PROGRAM TestsBase
VAR
	CyclicRunner_TEST			   : CyclicRunner_TEST;
	ComponentCollection_TEST	   : ComponentCollection_TEST;
	Module_TEST					   : Module_TEST;
	CyclicComponent_TEST		   : CyclicComponent_TEST;
	Component_TEST				   : Component_TEST;
	ModuleCollection_TEST		   : ModuleCollection_TEST;
	Tracing_TEST				   : Tracing_TEST;
	Initializer_TEST			   : Initializer_TEST;
	Events_TEST					   : Events_TEST;
	Statemachine_TEST			   : Statemachine_TEST;
	Collection_Test				   : Collection_TEST();
	List_TEST					   : List_TEST;
	ModeControl_TEST			   : ModeControl_TEST;
	CollectionPeeker_Test		   : CollectionPeeker_Test;
	ForcibleBool_TEST			   : ForcibleBool_TEST;
	ForcibleInt_Test			   : ForcibleInt_Test;
	Utilities_TEST				   : Utilities_TEST;
	DigitalInput_NC_TEST		   : DigitalInput_NC_TEST;
	DigitalInput_NO_TEST		   : DigitalInput_NO_TEST;
	DigitalOutput_TEST			   : DigitalOutput_TEST;
	DigitalInput_Combiner_TEST	   : DigitalInput_Combiner_TEST;
	DigitalInput_Debounce_TEST	   : DigitalInput_Debounce_TEST;
	Cylinder_TEST				   : Cylinder_TEST;
	SafetyBase_TEST				   : SafetyBase_TEST;
	ADS_TEST					   : ADS_TEST;
	DigitalInput_ForceVisitor_TEST : DigitalInput_ForceVisitor_TEST;
	Recipe_TEST					   : Recipe_TEST;
	Analog_TEST					   : Analog_TEST;
	Serial_TEST					   : SerialConnection_Tests;
	Axis_Test					   : Axis_Test;
	EtherCatMaster_TEST		   : EtherCatMaster_TEST;

	//
	Component1				  : CyclicComponent_Mockup('Component 1');
	Component2				  : CyclicComponent_Mockup('Component 2');
	Component3				  : CyclicComponent_Mockup('Component 3');
	Component4				  : CyclicComponent_Mockup('Component 4');
	Em						  : EquipmentModule_Mockup('Em', Component1, Component2);
	EmEm					  : MachineModule_Mockup('EmEm', Em, Component3, Component4);
	EmEmEm					  : MachineModule_Mockup('EmEmEm', EmEm, Component3, Component4);
	Machine					  : MachineModule_Mockup('Machine', EmEmEm, Component3, Component4);
	StringCollection		  : StringCollection<100>;
	MachineModuleVisitor	  : GetSystemTreeNamesVisitor(StringCollection);
	QueryInterfaceResettables : QueryInterfaceResettables();
	Rerun					  : BOOL;
END_VAR

GlobalTestSuite.TestSuite.TestSuiteName := 'Application Base Test Suite';
Tracing_TEST();
CyclicRunner_TEST();
ComponentCollection_TEST();
Module_TEST();
Component_TEST();
CyclicComponent_TEST();
ModuleCollection_TEST();
Initializer_TEST();
Events_TEST();
Statemachine_TEST();
Collection_Test();
List_TEST();
ModeControl_TEST();
CollectionPeeker_Test();
ForcibleBool_TEST();
Utilities_TEST();
DigitalInput_NC_TEST();
DigitalInput_NO_TEST();
DigitalOutput_TEST();
DigitalInput_Combiner_TEST();
DigitalInput_Debounce_TEST();
Cylinder_TEST();
SafetyBase_TEST();
ADS_TEST();
DigitalInput_ForceVisitor_TEST();
Recipe_TEST();
Analog_TEST();
AnyBuffer_TEST();
ForcibleInt_Test();
Serial_TEST();
Axis_Test();
EtherCatMaster_TEST();

// Mockup code
Samples_AnyBuffer();
//
IF NOT Machine.Initialized THEN
	Machine.Initialize();
ELSE
	Machine.CyclicLogic();
	MachineModuleVisitor.GetTree(Machine);
	QueryInterfaceResettables.GetAllResetComponents(Em);
END_IF

IF Rerun THEN
	Rerun := FALSE;
	GlobalTestSuite.TestSuite.ReRunTests();
END_IF

END_PROGRAM

(* stored: Version 1.1.0.1, ProductVersion 3.1.4026.18
   POU TestsBase: Id {9cddac07-df1f-4e43-80ae-f6917cc2c1c0}, SpecialFunc None *)
